FUNCTION_BLOCK Home extends CraneMovement
VAR_INPUT
END_VAR
VAR_OUTPUT
END_VAR
VAR
END_VAR

END_FUNCTION_BLOCK

(* stored: Version 1.1.0.1, ProductVersion 3.1.4024.10
   POU Home: Id {fff73924-f1b4-4ca9-b7bd-6e210259384d}, SpecialFunc None *)
